PROGRAM MeasureVariance
VAR
	// Inputs
	vXFromMotor AT%I*: LREAL;
	vYFromMotor AT%I*: LREAL;
	vThetaFromMotor AT%I*: LREAL;
	
	//Outputs
	v AT%Q*: LREAL;
	
	//local
	state: INT := 0;
	counter: INT := 0;
	
	//Odometry
	distX, distY, distTheta :LREAL :=0;
	// Task Freqeuncy in ms
	taskfreq: LREAL := 10;
	
	//the actual robot has to be selected in connecting PlcTaskInputs to actual Robot Camera data
	// x Koordinate bei Start nach Kamera
	camX AT%I*: LREAL := 0;
	// y Koordinate bei Start laut Kamera
	camY AT%I*: LREAL;
	// theta laut Kamera zu Beginn
	camTheta AT%I*: LREAL := 0;
	
	// Error in x
	ErrX: LREAL;
	// Error in y
	ErrY: LREAL;
	// Error in Theta
	ErrTheta: LREAL;
	//errorcam via UDP
	ErrCam AT%I*: LREAL;
	// soll geschwindigkeit
	vSoll: LREAL := 3;
END_VAR

(*IF state = 0 THEN
	v := 100;
	counter := counter+1;
	IF counter >  1990 THEN
		state:=1;
	END_IF
END_IF
	
IF state = 1 THEN
		v := 0;
END_IF *)

//state 0 to wait for cameraposition data
IF state = 0 THEN
	counter := counter+1;
	IF counter > 199 THEN
		state := 1;
		counter := 0;
	END_IF
END_IF

IF state = 1 THEN
	v := vSoll;
	
	
	//Initiale Pose nach Kamera als Startpose setzen
	IF counter < 1 THEN
		distX:= camX ;
		distY :=camY ;
		distTheta :=camTheta ;
	END_IF

	counter := counter + 1;
	IF counter > 199 THEN
		state := 2;
		counter := 0;
	END_IF
END_IF

IF state = 2 THEN
	v := 0;
	counter := counter + 1;
	IF counter > 199 THEN
		state := 3;
		counter := 0;
	END_IF
END_IF

IF state = 3 THEN
	v := vSoll;
	counter := counter + 1;
	IF counter > 199 THEN
		state := 4;
		counter := 0;
	END_IF
END_IF

IF state = 4 THEN
	v := 0;
END_IF

//Odometry calculation
distX := distX + vXFromMotor*taskfreq/1000;
distY := distY + vYFromMotor*taskfreq/1000;
distTheta := distTheta + vThetaFromMotor*taskfreq/1000;

//Error Calculation
ErrX := camX-distX; 
ErrY := camY-distY;
ErrTheta := camTheta-distTheta;

//ACHTUNG LOKALE ROBOTER DATEN MÜSSEN FÜR DIREKTE VERGLEICHBARKEI MIT KAMERAPOSE IN GLOBALE KS TRANSFORMEIRT WERDEN

END_PROGRAM

(* stored: Version 1.1.0.1, ProductVersion 3.1.4024.11
   POU MeasureVariance: Id {c75a3bf3-5869-4786-b230-7494e1c7eff4}, SpecialFunc None *)
